// Mitsubishi GX Works2 project: AGV_IOCHECK   PLC: Q03UD

PROGRAM MAIN
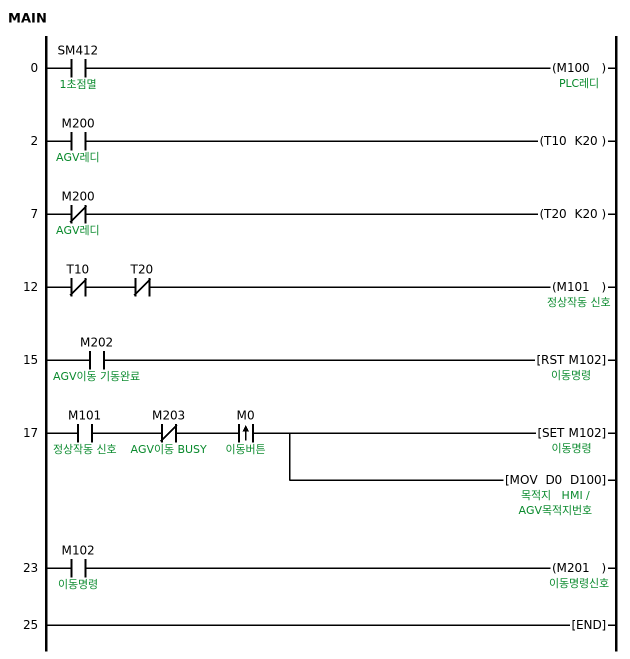
0     LD      SM412  ; 1초점멸
      OUT     M100  ; PLC레디
2     LD      M200  ; AGV레디
      OUT     T10 K20
7     LDI     M200  ; AGV레디
      OUT     T20 K20
12    LDI     T10
      ANI     T20
      OUT     M101  ; 정상작동 신호
15    LD      M202  ; AGV이동 기동완료
      RST     M102  ; 이동명령
17    LD      M101  ; 정상작동 신호
      ANI     M203  ; AGV이동 BUSY
      ANDP    M0  ; 이동버튼
      SET     M102  ; 이동명령
      MOV     D0 D100  ; 목적지   HMI / AGV목적지번호
23    LD      M102  ; 이동명령
      OUT     M201  ; 이동명령신호
25    END
END_PROGRAM
